FUNCTION_BLOCK TcoDesignerRootContainer EXTENDS TcoCore.TcoObject
VAR_INPUT
END_VAR
VAR_OUTPUT
END_VAR
VAR
END_VAR

END_FUNCTION_BLOCK

(* stored: Version 1.1.0.1, ProductVersion 3.1.4024.12
   POU TcoDesignerRootContainer: Id {c9188920-8b6d-08c2-3cbd-8695167d7e4d}, SpecialFunc None *)
